FUNCTION_BLOCK AGGREGATING (* Basic FB with empty ECC *)
  (* Standard: 61499-2 *)
  (* Version 1.0, 2020-10-21, chong *)
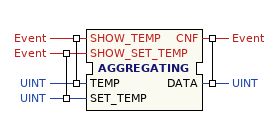
  EVENT_INPUT
    SHOW_TEMP WITH TEMP;
    SHOW_SET_TEMP WITH SET_TEMP;
  END_EVENT
  EVENT_OUTPUT
    CNF WITH DATA;
  END_EVENT
  VAR_INPUT
    TEMP : UINT;
    SET_TEMP : UINT;
  END_VAR
  VAR_OUTPUT
    DATA : UINT;
  END_VAR
  EC_STATES
    START; (* Initial State *)
  END_STATES
END_FUNCTION_BLOCK
